Yaskawa INFORM job: TEST_BP.JBI

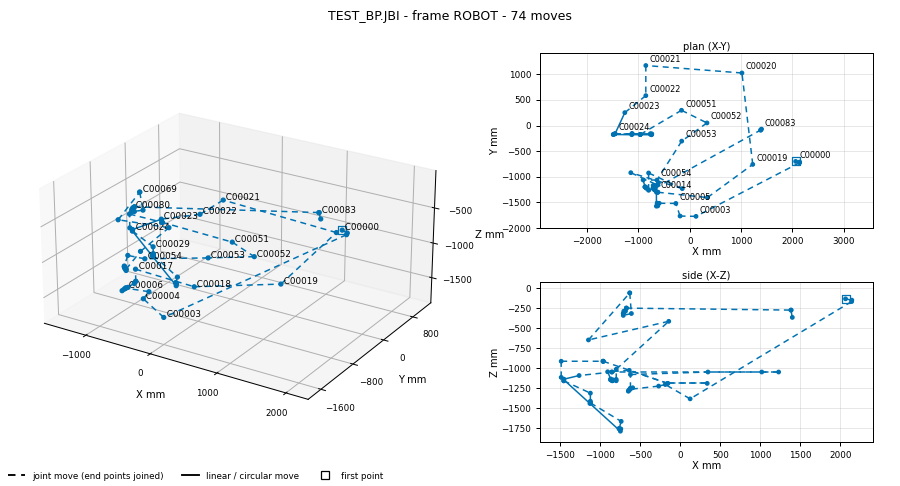
[picture p0: tool path of TEST_BP.JBI in frame ROBOT, 74 of 76 moves have a stored position in this frame; points joined in program order, loops and branches not executed]
/JOB
//NAME TEST_BP
//POS
///NPOS 86,86,76,5,0,0
///TOOL 0
///POSTYPE ROBOT
///RECTAN
///RCONF 0,0,0,0,1,0,0,0,0,0,0,0,0,0,0,0,0,0,0,0,0,0,0,0
C00000=2065.609,-700.442,-130.324,1.6821,-19.8072,-6.7552
///RCONF 0,0,0,0,0,0,0,0,0,0,0,0,0,0,0,0,0,0,0,0,0,0,0,0
C00001=2143.773,-711.949,-146.344,-1.3841,60.6353,174.7939
C00002=2141.712,-726.026,-164.078,-20.6195,56.8864,145.1128
C00003=121.874,-1771.649,-1380.986,36.5382,6.1742,118.9307
C00004=-188.884,-1765.779,-1201.769,36.5382,6.1757,108.8890
C00005=-271.321,-1519.419,-1221.579,44.4105,29.4004,111.1614
C00006=-633.316,-1516.391,-1262.220,53.2467,12.5433,98.9174
C00007=-633.297,-1516.757,-1290.102,53.2461,12.5433,98.9191
C00008=-633.316,-1516.391,-1262.220,53.2467,12.5433,98.9174
C00009=-651.556,-1516.370,-1262.237,53.2460,12.5449,98.9145
C00010=-633.314,-1516.366,-1262.246,53.2462,12.5415,98.9173
C00011=-596.638,-1516.332,-1242.131,53.2598,12.5355,98.9202
C00012=-624.101,-1568.002,-1256.059,44.4078,29.3892,111.1662
C00013=-651.001,-1572.920,-1281.021,44.4033,29.3920,111.1598
C00014=-649.684,-1300.988,-1284.705,44.4027,29.3874,111.1616
C00015=-624.553,-1300.993,-1248.861,44.4038,29.3836,111.1658
C00016=-624.562,-1300.989,-1248.860,44.4041,29.3835,111.1655
C00017=-624.556,-1300.988,-1076.871,44.4037,29.3823,111.1669
C00018=344.573,-1405.060,-1045.323,45.1904,30.5203,150.9270
C00019=1228.518,-758.439,-1045.323,45.1904,30.5203,-164.6188
C00020=1017.775,1024.641,-1045.323,45.1904,30.5203,-87.9642
C00021=-856.927,1169.934,-1045.323,45.1904,30.5203,-6.9633
C00022=-856.917,582.723,-1045.332,45.1901,30.5197,-6.9637
///RCONF 1,0,0,0,1,0,0,0,0,0,0,0,0,0,0,0,0,0,0,0,0,0,0,0
C00023=-1266.536,251.157,-1089.460,29.2167,46.4569,29.6919
///RCONF 0,0,0,0,0,0,0,0,0,0,0,0,0,0,0,0,0,0,0,0,0,0,0,0
C00024=-1456.148,-160.344,-1134.660,58.6699,26.1984,120.0642
C00025=-1458.498,-161.490,-1171.147,58.6659,26.1967,120.0677
C00026=-1458.548,-161.340,-1155.382,58.6616,26.1901,120.0553
C00027=-1458.550,-187.806,-1155.364,58.6614,26.1877,120.0552
C00028=-1458.551,-161.334,-1155.380,58.6620,26.1901,120.0550
C00029=-1125.633,-162.687,-1309.436,58.6580,26.1872,120.0590
C00030=-1125.640,-162.684,-1410.229,58.6582,26.1861,120.0594
C00031=-1125.594,-162.711,-1431.396,58.6560,26.1865,120.0607
C00032=-1125.589,-162.720,-1453.074,58.6564,26.1897,120.0595
C00033=-1125.594,-162.711,-1431.396,58.6560,26.1865,120.0607
C00034=-1125.604,-191.683,-1431.389,58.6563,26.1865,120.0597
C00035=-1125.594,-162.711,-1431.396,58.6560,26.1865,120.0607
C00036=-740.157,-162.726,-1662.593,58.6563,26.1862,120.0624
///RCONF 0,0,0,0,1,0,0,0,0,0,0,0,0,0,0,0,0,0,0,0,0,0,0,0
C00037=-765.739,-164.955,-1753.345,58.6544,26.1855,120.0613
C00038=-765.755,-164.961,-1776.727,58.6558,26.1826,120.0644
C00039=-765.739,-164.955,-1753.345,58.6544,26.1855,120.0613
C00040=-765.723,-194.487,-1753.340,58.6547,26.1879,120.0628
C00041=-765.739,-164.955,-1753.345,58.6544,26.1855,120.0613
C00042=-744.950,-179.324,-1756.566,58.6516,26.1799,120.0614
C00043=-750.107,-179.323,-1785.497,58.6533,26.1800,120.0623
///RCONF 0,0,0,0,0,0,0,0,0,0,0,0,0,0,0,0,0,0,0,0,0,0,0,0
C00044=-1131.380,-179.374,-1438.769,58.6549,26.1820,120.0657
C00045=-1490.588,-175.163,-1112.451,58.6559,26.1849,120.0660
C00046=-1490.601,-175.164,-910.781,58.6568,26.1847,120.0664
C00047=-965.795,-175.163,-910.787,58.6563,26.1850,120.0665
C00048=-965.795,-175.163,-910.787,58.6563,26.1850,120.0665
C00049=-965.803,-175.270,-910.733,58.6655,26.1971,120.0700
C00050=-965.803,-175.270,-910.733,58.6655,26.1971,120.0700
C00051=-160.460,296.677,-1187.553,4.5148,32.7346,67.8388
C00052=335.614,50.286,-1187.553,4.5148,32.7346,-41.3584
C00053=-156.788,-304.212,-1187.553,4.5148,32.7346,-167.8326
C00054=-639.174,-1064.987,-1024.365,14.9351,29.3158,-160.1089
C00055=-909.494,-1061.541,-1042.262,2.0196,6.1445,-137.3260
C00056=-871.852,-1197.994,-1131.945,2.2539,4.0308,-137.3045
C00057=-871.853,-1197.992,-1142.507,2.2540,4.0306,-137.3055
C00058=-871.872,-1197.959,-1153.569,2.2488,4.0298,-137.2965
C00059=-871.853,-1197.992,-1142.507,2.2540,4.0306,-137.3055
C00060=-847.083,-1219.883,-1142.524,2.2529,4.0307,-137.3022
C00061=-847.084,-1219.882,-1154.733,2.2529,4.0305,-137.3025
C00062=-855.432,-1204.525,-1154.750,2.2513,4.0316,-137.3003
C00063=-810.212,-1207.678,-1154.782,2.2489,4.0315,-137.3008
C00064=-802.438,-1259.228,-1154.780,2.2485,4.0311,-137.3005
C00065=-802.435,-1259.230,-1137.498,2.2486,4.0314,-137.2999
C00066=-802.403,-925.593,-1011.044,2.2476,4.0354,-137.2976
C00067=-145.318,-1230.412,-411.342,-92.0451,29.6168,34.4172
C00068=-1149.668,-920.379,-644.277,-120.1740,-14.5460,-53.6729
C00069=-633.345,-1159.538,-56.519,179.0503,43.9245,-118.1181
C00070=-633.345,-1159.538,-56.519,179.0503,43.9245,-118.1181
C00071=-612.676,-1123.690,-313.661,179.7932,56.6722,-117.5430
C00072=-713.698,-1170.858,-337.488,-179.8412,57.7313,-117.2352
C00073=-713.708,-1221.257,-314.263,-179.8466,57.7304,-117.2406
C00074=-713.708,-1221.257,-314.263,-179.8466,57.7304,-117.2406
C00075=-721.684,-1229.153,-314.260,-179.8452,57.7299,-117.2415
C00076=-713.708,-1221.257,-314.263,-179.8466,57.7304,-117.2406
C00077=-686.695,-1255.029,-284.714,-179.8476,57.7296,-117.2417
///RCONF 1,0,0,0,0,0,0,0,0,0,0,0,0,0,0,0,0,0,0,0,0,0,0,0
C00078=-707.334,-1236.789,-284.690,-179.8481,57.7287,-117.2422
C00079=-691.430,-1243.701,-253.740,-179.8706,57.7317,-117.2644
///RCONF 0,0,0,0,0,0,0,0,0,0,0,0,0,0,0,0,0,0,0,0,0,0,0,0
C00080=-675.419,-1259.857,-246.458,-179.8615,57.7244,-117.2555
///RCONF 1,0,0,0,0,0,0,0,0,0,0,0,0,0,0,0,0,0,0,0,0,0,0,0
C00081=-675.408,-1222.263,-246.433,-179.8615,57.7235,-117.2550
C00082=-675.408,-1222.263,-246.433,-179.8615,57.7235,-117.2550
C00083=1385.216,-87.208,-270.968,-179.8598,57.7242,-2.4475
C00084=1382.202,-90.184,-270.996,-179.8607,57.7243,-2.4486
C00085=1399.685,-70.079,-362.341,65.8103,-64.9357,-61.8468
///RCONF 0,0,0,0,0,0,0,0,0,0,0,0,0,0,0,0,0,0,0,0,0,0,0,0
BC00000=786.422,3373.682,1399.077
BC00001=786.422,3373.676,1057.321
BC00002=1256.493,3266.508,860.929
BC00003=2201.430,3266.508,860.929
BC00004=2278.176,2275.411,570.669
BC00005=2443.660,2275.411,570.669
BC00006=2443.660,2275.411,570.669
BC00007=2443.654,2275.418,570.656
BC00008=2443.660,2275.411,570.669
BC00009=2443.660,2275.411,570.669
BC00010=2443.660,2275.418,570.664
BC00011=2443.660,2275.424,570.658
BC00012=2443.654,2275.424,570.645
BC00013=2443.654,2275.424,570.645
BC00014=2443.654,2275.431,570.634
BC00015=2443.654,2275.431,570.628
BC00016=2443.654,2275.431,717.005
BC00017=2443.654,1995.448,787.684
BC00018=2443.654,1995.461,1148.378
BC00019=2430.426,1347.032,1148.378
BC00020=2430.426,772.016,1148.378
BC00021=2430.426,772.016,1148.378
BC00022=2430.426,772.016,1148.378
BC00023=2430.426,772.016,1148.378
BC00024=2430.438,1190.603,1148.365
BC00025=2430.438,1190.603,1148.354
BC00026=2430.438,1190.603,1148.371
BC00027=2430.438,1190.603,1148.371
BC00028=2430.438,1190.603,1148.371
BC00029=2430.438,1190.603,1148.360
BC00030=2430.438,1190.603,1148.360
BC00031=2430.438,1190.603,1148.354
BC00032=2430.438,1190.603,1148.354
BC00033=2430.438,1190.603,1148.354
BC00034=2430.438,1190.603,1148.354
BC00035=2430.438,1190.603,1148.354
BC00036=2430.438,1190.603,1148.354
BC00037=2430.438,1190.603,1148.354
BC00038=2430.438,1190.603,1148.354
BC00039=2430.438,1190.603,1148.354
BC00040=2430.438,1190.603,1148.354
BC00041=2430.438,1190.603,1148.354
BC00042=2430.445,1190.603,1148.347
BC00043=2430.445,1190.603,1148.347
BC00044=2430.445,1190.603,1148.347
BC00045=2430.445,1190.603,1148.347
BC00046=2430.445,1190.603,1148.347
BC00047=2430.445,1190.603,1148.347
BC00048=2454.428,3687.445,1148.347
BC00049=2454.428,3687.439,1148.345
BC00050=2454.428,1365.683,1148.345
BC00051=2454.428,1365.683,1148.345
BC00052=2454.428,1365.683,1148.345
BC00053=2454.428,1365.683,1148.345
BC00054=2454.428,1365.683,1148.345
BC00055=2454.428,1365.683,1148.345
BC00056=2454.428,1365.683,1148.345
BC00057=2454.428,1365.683,1148.345
BC00058=2454.428,1365.683,1148.345
BC00059=2454.428,1365.683,1148.345
BC00060=2454.428,1365.689,1148.339
BC00061=2454.428,1365.689,1148.339
BC00062=2454.428,1365.689,1148.339
BC00063=2454.428,1365.689,1148.339
BC00064=2454.428,1365.689,1148.339
BC00065=2454.428,1365.689,1148.339
BC00066=2454.428,1948.251,1148.335
BC00067=2454.428,1948.251,1148.335
BC00068=2437.639,1747.697,1041.254
BC00069=2437.639,1751.941,1041.254
BC00070=2437.639,1632.033,66.583
BC00071=2437.639,1500.453,66.583
BC00072=2437.639,1506.221,66.583
BC00073=2437.639,1506.221,66.583
BC00074=2437.639,1506.221,66.583
BC00075=2437.639,1506.221,66.583
BC00076=2437.639,1506.221,66.583
BC00077=2437.639,1506.221,66.583
BC00078=2437.639,1506.221,66.583
BC00079=2437.639,1506.221,66.583
BC00080=2437.639,1506.221,66.583
BC00081=2437.639,1506.221,66.583
BC00082=2437.639,2440.108,66.583
BC00083=2437.639,2440.108,66.583
BC00084=2218.193,3322.969,66.583
BC00085=783.999,3555.357,1358.398
///POSTYPE PULSE
///PULSE
EC00000=-1,1
EC00001=-2,1
EC00002=-1,1
EC00003=-1,1
EC00004=-1,1
EC00005=-1,1
EC00006=-1,1
EC00007=-1,1
EC00008=-1,1
EC00009=-1,1
EC00010=-2,1
EC00011=-2,1
EC00012=-2,1
EC00013=-2,1
EC00014=-2,1
EC00015=-2,1
EC00016=-2,1
EC00017=-2,1
EC00018=-2,1
EC00019=-2,1
EC00020=-2,1
EC00021=-2,1
EC00022=-2,1
EC00023=-2,1
EC00024=-2,1
EC00025=-2,1
EC00026=-2,1
EC00027=-2,1
EC00028=-2,1
EC00029=-2,1
EC00030=-2,1
EC00031=-2,1
EC00032=-2,1
EC00033=-2,1
EC00034=-1,0
EC00035=-1,0
EC00036=-1,0
EC00037=-1,0
EC00038=-1,0
EC00039=-1,0
EC00040=-1,0
EC00041=-566918,-177956
EC00042=-566918,-177956
EC00043=-566918,-177956
EC00044=-566918,-177956
EC00045=-566918,-177956
EC00046=-566918,-177956
EC00047=-566918,-177956
EC00048=-566918,-177956
EC00049=-566918,-177956
EC00050=-566918,-177956
EC00051=-566917,-177956
EC00052=-566917,-177956
EC00053=-566917,-177956
EC00054=-566917,-177956
EC00055=-566917,-177956
EC00056=-566917,-177956
EC00057=-566917,-177956
EC00058=-566917,-177956
EC00059=-566917,-177956
EC00060=-566917,-177956
EC00061=-566917,-177956
EC00062=-566917,-177956
EC00063=-566917,-177956
EC00064=-566917,-177956
EC00065=-566917,-177956
EC00066=-566917,-177956
EC00067=-566917,-177956
EC00068=-566917,-177956
EC00069=-566917,-177956
EC00070=-566917,-177956
EC00071=-566917,-177956
EC00072=-566917,-177956
EC00073=-566917,-177956
EC00074=-566917,-177956
EC00075=-566917,-177956
///POSTYPE BASE
///RECTAN
///RCONF 0,0,0,0,1,0,0,0,0,0,0,0,0,0,0,0,0,0,0,0,0,0,0,0
P00006=2.006,1.622,-0.565,0.0000,0.0000,0.0000
///RCONF 0,0,0,0,0,0,0,0,0,0,0,0,0,0,0,0,0,0,0,0,0,0,0,0
P00040=2.716,-0.016,3.014,0.0000,0.0000,0.0000
P00041=-0.109,0.014,0.966,0.0000,0.0000,0.0000
P00042=-0.220,0.371,-0.613,0.0000,0.0000,0.0000
P00043=-0.179,-5.890,-3.227,0.0000,0.0000,0.0000
//INST
///DATE 2024/01/23 15:58
///ATTR SC,RW,RJ
////FRAME ROBOT
///GROUP1 RB1,BS1
///GROUP2 ST1
NOP
SFTOF
CALL JOB:CLEAN-R1_LONG
SFTOF
MOVJ C00000 BC00000 VJ=100.00  +MOVJ EC00000 VJ=0.78
MOVJ C00001 BC00001 VJ=100.00  +MOVJ EC00001 VJ=100.00
MOVJ C00002 BC00002 VJ=100.00  +MOVJ EC00002 VJ=0.78
MOVJ C00003 BC00003 VJ=100.00  +MOVJ EC00003 VJ=100.00
MOVJ C00004 BC00004 VJ=100.00  +MOVJ EC00004 VJ=100.00
MOVJ C00005 BC00005 VJ=100.00  +MOVJ EC00005 VJ=100.00
SFTOF
MOVJ C00006 BC00006 VJ=100.00  +MOVJ EC00006 VJ=100.00
REFP 3 RB1 C00007 BC00007
CALL JOB:SEARCH-R1
SET P040 P006
SFTON P040
MOVJ C00008 BC00008 VJ=100.00  +MOVJ EC00007 VJ=0.78
REFP 3 RB1 C00009 BC00009
CALL JOB:SEARCH-R1
SET P040 P006
SFTON P040
MOVJ C00010 BC00010 VJ=100.00  +MOVJ EC00008 VJ=100.00
MOVJ C00011 BC00011 VJ=100.00  +MOVJ EC00009 VJ=0.78
SFTOF
MACRO1 MJ#(0) ARGF9
SFTON P040
MOVJ C00012 BC00012 VJ=100.00  +MOVJ EC00010 VJ=100.00
MOVJ C00013 BC00013 VJ=20.00  +MOVJ EC00011 VJ=100.00
ARCON
MOVL C00014 BC00014 V=11.0  +MOVJ EC00012 VJ=20.00
ARCOF
MOVJ C00015 BC00015 VJ=100.00  +MOVJ EC00013 VJ=20.00
MOVJ C00016 BC00016 VJ=100.00  +MOVJ EC00014 VJ=0.78
MOVJ C00017 BC00017 VJ=100.00  +MOVJ EC00015 VJ=0.78
MOVJ C00018 BC00018 VJ=100.00  +MOVJ EC00016 VJ=100.00
MOVJ C00019 BC00019 VJ=100.00  +MOVJ EC00017 VJ=100.00
MOVJ C00020 BC00020 VJ=100.00  +MOVJ EC00018 VJ=100.00
MOVJ C00021 BC00021 VJ=100.00  +MOVJ EC00019 VJ=100.00
MOVJ C00022 BC00022 VJ=100.00  +MOVJ EC00020 VJ=100.00
MOVJ C00023 BC00023 VJ=100.00  +MOVJ EC00021 VJ=100.00
SFTOF
MOVL C00024 BC00024 V=83.3  +MOVJ EC00022 VJ=100.00
REFP 3 RB1 C00025 BC00025
CALL JOB:SEARCH-R1
SET P041 P006
SFTON P041
MOVJ C00026 BC00026 VJ=100.00  +MOVJ EC00023 VJ=0.78
REFP 3 RB1 C00027 BC00027
CALL JOB:SEARCH-R1
SET P041 P006
SFTON P041
MOVJ C00028 BC00028 VJ=100.00  +MOVJ EC00024 VJ=100.00
SFTOF
MOVJ C00029 BC00029 VJ=100.00  +MOVJ EC00025 VJ=100.00
MOVJ C00030 BC00030 VJ=100.00  +MOVJ EC00026 VJ=0.78
MOVL C00031 BC00031 V=83.3  +MOVJ EC00027 VJ=100.00
REFP 3 RB1 C00032 BC00032
CALL JOB:SEARCH-R1
SET P042 P006
SFTON P042
MOVJ C00033 BC00033 VJ=100.00  +MOVJ EC00028 VJ=0.78
REFP 3 RB1 C00034 BC00034
CALL JOB:SEARCH-R1
SET P042 P006
SFTON P042
MOVJ C00035 BC00035 VJ=100.00  +MOVJ EC00029 VJ=100.00
MOVJ C00036 BC00036 VJ=100.00  +MOVJ EC00030 VJ=100.00
SFTOF
MOVL C00037 BC00037 V=83.3  +MOVJ EC00031 VJ=100.00
REFP 3 RB1 C00038 BC00038
CALL JOB:SEARCH-R1
SET P043 P006
SFTON P043
MOVJ C00039 BC00039 VJ=100.00  +MOVJ EC00032 VJ=0.78
REFP 3 RB1 C00040 BC00040
CALL JOB:SEARCH-R1
SET P043 P006
SFTON P043
MOVJ C00041 BC00041 VJ=100.00  +MOVJ EC00033 VJ=100.00
SFTOF
MOVJ C00042 BC00042 VJ=100.00  +MOVJ EC00034 VJ=100.00
MACRO1 MJ#(0) ARGF9
SFTON P043
MOVL C00043 BC00043 V=11.0  +MOVJ EC00035 VJ=100.00
ARCON
MOVL C00044 BC00044 V=11.0  +MOVJ EC00036 VJ=100.00
SFTON P042
MOVL C00045 BC00045 V=11.0  +MOVJ EC00037 VJ=100.00
ARCOF
MOVJ C00046 BC00046 VJ=100.00  +MOVJ EC00038 VJ=100.00
MOVJ C00047 BC00047 VJ=100.00  +MOVJ EC00039 VJ=0.78
MOVJ C00048 BC00048 VJ=100.00  +MOVJ EC00040 VJ=100.00
MOVJ C00049 BC00049 VJ=100.00  +MOVJ EC00041 VJ=100.00
MOVJ C00050 BC00050 VJ=100.00  +MOVJ EC00042 VJ=100.00
MOVJ C00051 BC00051 VJ=100.00  +MOVJ EC00043 VJ=100.00
MOVJ C00052 BC00052 VJ=100.00  +MOVJ EC00044 VJ=100.00
MOVJ C00053 BC00053 VJ=100.00  +MOVJ EC00045 VJ=100.00
MOVJ C00054 BC00054 VJ=100.00  +MOVJ EC00046 VJ=100.00
MOVJ C00055 BC00055 VJ=100.00  +MOVJ EC00047 VJ=100.00
SFTOF
MOVJ C00056 BC00056 VJ=100.00  +MOVJ EC00048 VJ=100.00
MOVJ C00057 BC00057 VJ=100.00  +MOVJ EC00049 VJ=100.00
REFP 3 RB1 C00058 BC00058
CALL JOB:SEARCH-R1
SET P043 P006
SFTON P043
MOVJ C00059 BC00059 VJ=100.00  +MOVJ EC00050 VJ=0.78
MOVJ C00060 BC00060 VJ=100.00  +MOVJ EC00051 VJ=100.00
MOVJ C00061 BC00061 VJ=100.00  +MOVJ EC00052 VJ=100.00
MOVC C00062 BC00062 V=11.0  +MOVJ EC00053 VJ=100.00
MOVC C00063 BC00063 V=11.0  +MOVJ EC00054 VJ=100.00
MOVC C00064 BC00064 V=11.0  +MOVJ EC00055 VJ=100.00
MOVJ C00065 BC00065 VJ=100.00  +MOVJ EC00056 VJ=100.00
SFTOF
MOVJ C00066 BC00066 VJ=100.00  +MOVJ EC00057 VJ=100.00
MOVJ C00067 BC00067 VJ=100.00  +MOVJ EC00058 VJ=100.00
MOVJ C00068 BC00068 VJ=100.00  +MOVJ EC00059 VJ=100.00
MOVJ C00069 BC00069 VJ=100.00  +MOVJ EC00060 VJ=100.00
MOVJ C00070 BC00070 VJ=100.00  +MOVJ EC00061 VJ=100.00
MOVJ C00071 BC00071 VJ=100.00  +MOVJ EC00062 VJ=100.00
MOVJ C00072 BC00072 VJ=100.00  +MOVJ EC00063 VJ=100.00
MOVJ C00073 BC00073 VJ=100.00  +MOVJ EC00064 VJ=100.00
SFTOF
MOVJ C00074 BC00074 VJ=100.00  +MOVJ EC00065 VJ=100.00
REFP 3 RB1 C00075 BC00075
CALL JOB:SEARCH-R1
SET P043 P006
SFTON P043
MOVJ C00076 BC00076 VJ=100.00  +MOVJ EC00066 VJ=0.78
MOVJ C00077 BC00077 VJ=100.00  +MOVJ EC00067 VJ=100.00
MOVC C00078 BC00078 V=11.0  +MOVJ EC00068 VJ=100.00
MOVC C00079 BC00079 V=11.0  +MOVJ EC00069 VJ=100.00
MOVC C00080 BC00080 V=11.0  +MOVJ EC00070 VJ=100.00
MOVJ C00081 BC00081 VJ=100.00  +MOVJ EC00071 VJ=100.00
MOVJ C00082 BC00082 VJ=100.00  +MOVJ EC00072 VJ=100.00
MOVJ C00083 BC00083 VJ=100.00  +MOVJ EC00073 VJ=100.00
SFTOF
MOVJ C00084 BC00084 VJ=100.00  +MOVJ EC00074 VJ=100.00
MOVJ C00085 BC00085 VJ=100.00  +MOVJ EC00075 VJ=100.00
CALL JOB:0_0
CALL JOB:CLEAN-R1_LONG
END
